Universal Robots PolyScope program: Weight_Train.urp

Program Weight_Train (installation=default directory=/programs/usbdisk_0/new folder createdIn=5.8.0.10253 lastSavedIn=5.8.0.10253 robotSerialNumber=20205300708)
Calibrated DH parameters: a=[-0.000048, -0.164988, -0.190768, -0.000044, -0.000167, 0]; d=[0.151937, 265.766517, -282.786649, 17.1509, 0.085408, 0.091845]; alpha=[1.570475, 0.000674, 0.005589, 1.571818, -1.57228, 0]; deltaTheta=[0, 0.826521, -1.289102, 0.462588, 0, 0]
BeforeStart
  weight := 9999
  MoveJ speed 60 deg/s, acceleration 80 deg/s^2 (useActiveTCP=true) feature=Base
    Waypoint grabPos: TCP in base x=353.876 y=-243.821 z=429.31 mm, rx=1.7497 ry=1.6183 rz=-0.8122 rad; joints [-6.519, -115.266, -35, -114.309, -320.921, -904.661] deg
  Popup Warning (haltProgram=false message=Gripper will open and potentially drop something inputType=Text)
  URCap Gripper Activate (Robotiq_Grippers, Robotiq Inc.) dataModel(ResetAndActivateKey=false)
  URCap Gripper (Robotiq_Grippers, Robotiq Inc.) dataModel(position=0.0, force=100.0, speed=100.0, positionInDouble=0.0, forceInDouble=100.0, speedInDouble=100.0, slaveIds=[9], blocking=true)
  Loop While (checkContinuously=false) expression=weight<0 or weight>6.6
    weight :=  (valueSource=Operator message=Input the weight of the object in lbs. valueType=Float)
    If weight≥0 and weight≤6.6
      Set ExpressionOutput pin=ObjectWeight; expression=weight*1000
    Else 
      Popup Message (haltProgram=false message=Weight must be between 0 - 6.6 inputType=Text)
  Popup Message (haltProgram=false message=Place object in gripper inputType=Text)
  Wait Sleep waitTime=1
  URCap Gripper (Robotiq_Grippers, Robotiq Inc.) dataModel(position=100.0, force=100.0, speed=100.0, positionInDouble=100.0, forceInDouble=100.0, speedInDouble=100.0, slaveIds=[9], blocking=true)
Robot Program (runOnlyOnce=false)
  MoveJ speed 60 deg/s, acceleration 80 deg/s^2 (useActiveTCP=true) feature=Base
    Waypoint WeighPoint: TCP in base x=-373.14 y=-331.845 z=292.511 mm, rx=0.6282 ry=1.4698 rz=-0.5607 rad; joints [-133.922, -144.995, -35.002, -90, -179.679, -1077.387] deg
    Wait Sleep waitTime=2
    Set ExpressionOutput pin=position; expression=1
    Wait Sleep waitTime=30
    Set ExpressionOutput pin=position; expression=0
    Wait Sleep waitTime=2
  MoveJ speed 60 deg/s, acceleration 80 deg/s^2 (useActiveTCP=true) feature=Base
    Waypoint grabPos: TCP in base x=353.876 y=-243.821 z=429.31 mm, rx=1.7497 ry=1.6183 rz=-0.8122 rad; joints [-6.519, -115.266, -35, -114.309, -320.921, -904.661] deg
  rmv_obj :=  (valueSource=Operator message=Remove object? valueType=Boolean)
  If rmv_obj≟ True
    URCap Gripper (Robotiq_Grippers, Robotiq Inc.) dataModel(position=0.0, force=100.0, speed=100.0, positionInDouble=0.0, forceInDouble=100.0, speedInDouble=100.0, slaveIds=[9], blocking=true)
    weight :=  (valueSource=Operator message=What is the weight of the object in lbs. valueType=Float)
    Set ExpressionOutput pin=ObjectWeight; expression=weight*1000
    Popup Message (haltProgram=false message=Place object in gripper inputType=Text)
    Wait Sleep waitTime=1
    URCap Gripper (Robotiq_Grippers, Robotiq Inc.) dataModel(position=100.0, force=100.0, speed=100.0, positionInDouble=100.0, forceInDouble=100.0, speedInDouble=100.0, slaveIds=[9], blocking=true)
